PROGRAM P_Demo_FB_LicFileCopyFromDongle
VAR
    fbFB_LicFileCopyFromDongle : FB_LicFileCopyFromDongle; // FB_LicFileCopyFromDongle 实例
    bExec                      : BOOL := FALSE;
    bBusy_                     : BOOL;
    bErrFlag                   : BOOL;
    nErrCode                   : UDINT;
END_VAR

// =============================================================================
// 场景：备份 dongle License。
// 价值：备份支持。
// 验证：触发后观察 bDone / bErr，错误号 nErrId 反映 ADS Return Codes。
// 验证步骤：
//   1. 右键 PLC 项目下 POUs 文件夹 → Add → Existing Item → 选本 .TcPOU 文件
//   2. 引用 Tc2_Utilities（References → Add library）
//   3. 编译 → 登录 → 运行；按上方『验证』行的指示在线写值观察
// =============================================================================

fbFB_LicFileCopyFromDongle(
    bExecute := bExec, tTimeout := DEFAULT_ADS_TIMEOUT,
    bBusy => bBusy_, bError => bErrFlag, nErrorId => nErrCode
);

END_PROGRAM

(* stored: Version 1.1.0.1, ProductVersion 3.1.4024.5
   POU P_Demo_FB_LicFileCopyFromDongle: Id {2f7609a0-dcb1-58d0-8966-e3fe803dadd6}, SpecialFunc None *)
